TYPE ST_FSoE_08Byte :
STRUCT
	CMD		: BYTE;
	SafeData1 	: WORD;
	CRC1		: WORD;
	SafeData2 	: WORD;
	CRC2		: WORD;
	SafeData3 	: WORD;
	CRC3		: WORD;
	SafeData4 	: WORD;
	CRC4		: WORD;
	ConnID		: WORD;
END_STRUCT
END_TYPE

(* stored: Version 1.1.0.1, ProductVersion 3.1.4024.5
   DUT ST_FSoE_08Byte: Id {f5ddda5e-12df-4bdb-b542-5268babd247b} *)
